TYPE ExerciseCirculationPumpsParameters :
STRUCT
	Interval: INT := 24; (* Central exercise interval for all damper modules (set to zero for no exercising) $(unit hour) *)
	StopVentilation: BOOL := FALSE; (* Stop ventilation during central exercise *)
	Hour: INT := 10; (* Central exercise at this hour $(unit hour) *)
	Minute: INT := 30; (* Central exercise at this minute $(unit minute) *)
	(*
	TimeChannel: TimeChannelSettings;
	StartManualExercise: BOOL;
	ExerciseStatus: BOOL;
	*)
END_STRUCT
END_TYPE

(* stored: Version 1.1.0.1, ProductVersion 3.1.4024.6
   DUT ExerciseCirculationPumpsParameters: Id {f77bbff2-c0d5-4208-9197-de5d53b514f7} *)
